FUNCTION FC3_Safety : BOOL
VAR_INPUT
END_VAR
VAR
END_VAR



IF  DB10_Alias.ix_E_stopNC AND NOT DB10_Alias.ix_E_stopNO THEN
	
	FC3_Safety := TRUE;
ELSE
	FC3_Safety := FALSE;
END_IF

END_FUNCTION

(* stored: Version 1.1.0.1, ProductVersion 3.1.4024.12
   POU FC3_Safety: Id {d8ed1706-68af-4960-a196-078473d8ccab}, SpecialFunc None *)
